FUNCTION_BLOCK CTRL_OUT (* Control Output with Limit and Manual Override *)
  (* Standard: 61499-1; Description: CTRL_OUT adds to the CI input the value of OFFSET and returns the result to Y if MANUAL = FALSE. If MANUAL is TRUE at output Y the input value of MAN_IN + OFFSET is issued. Y is always limited to the boundaries defined by LIM_L and LIM_H. If Y reaches one of the limits, then the output LIM is TRUE. CTRL_OUT can be used to build own rule modules. *)
  (* Version 1.1, 2008-11-05, oscat/hugo, Original TwinCAT Version *)
  (* Version 1.0, 2025-12-19, Franz Höpfinger, Converted to 4diac; initial API and implementation and/or initial documentation *)
  PACKAGE OSCAT::Basic::POUs::Engineering::Control;
  IMPORT eclipse4diac::core::TypeHash;
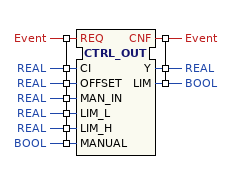
  EVENT_INPUT
    REQ WITH CI, OFFSET, MAN_IN, LIM_L, LIM_H, MANUAL; (* Normal Execution Request *)
  END_EVENT
  EVENT_OUTPUT
    CNF WITH Y, LIM; (* Execution Confirmation *)
  END_EVENT
  VAR_INPUT
    CI : REAL; (* Control Input *)
    OFFSET : REAL; (* Offset *)
    MAN_IN : REAL; (* Manual Input Value *)
    LIM_L : REAL; (* Low Limit *)
    LIM_H : REAL; (* High Limit *)
    MANUAL : BOOL; (* Manual Mode Active *)
  END_VAR
  VAR_OUTPUT
    Y : REAL; (* Control Output *)
    LIM : BOOL; (* Limit Reached Flag *)
  END_VAR
  EC_STATES
    REQ : REQ -> CNF;
  END_STATES
  ALGORITHM REQ IN ST:
(* Calculate Output based on Manual/Auto *)
Y := SEL(MANUAL, CI, MAN_IN) + OFFSET;

(* Limit the output *)
IF Y > LIM_L AND Y < LIM_H THEN
	LIM := FALSE;
ELSE
	Y := LIMIT(LIM_L, Y, LIM_H);
	LIM := TRUE;
END_IF;
  END_ALGORITHM
END_FUNCTION_BLOCK
